Staubli VAL3: refreshDynamic.pgx

program refreshDynamic()
begin
  // DO NOT CHANGE
  nRefresh=clock()
  use:bUseRefresh=false
  //
  // ADD HERE
  //
  call buildList()
  //
  // refresh the cursor
  use:nView=nView
  // refresh the list
  call use:listupdate(nIndex-nView)
end
